// TIA Portal V17 export
// export: Created 2023-02-14T02:49:55.0959699Z, ExportSetting WithDefaults, DisplayName Totally Integrated Automation Portal, DisplayVersion V17, DisplayName TIA Portal Openness, DisplayVersion V17, DisplayName TIA Portal Teamcenter Gateway, DisplayVersion V17, DisplayName TIA Portal Version Control Interface, DisplayVersion V17, DisplayName SINAMICS Startdrive Advanced, DisplayVersion V17, DisplayName SINAMICS Startdrive G130, G150, S120, S150, SINAMICS MV, S210, DisplayVersion V17, DisplayName SINAMICS Startdrive G110M, G120, G120C, G120D, G120P, G115D, DisplayVersion V17, DisplayName STEP 7 Professional, DisplayVersion V17, DisplayName STEP 7 Safety, DisplayVersion V17, DisplayName WinCC Professional, DisplayVersion V17
VAR_GLOBAL   // PLC tag table "RIO Preparation"
   "FT-51.01" AT %IW83 : Int;
   "TT-51.01" AT %IW85 : Int;
   "LT-02.01" AT %IW87 : Int;
   "LT-03.01" AT %IW89 : Int;
   "LT-04.01" AT %IW91 : Int;
   "LT-05.01" AT %IW93 : Int;
   "LT-06.01" AT %IW95 : Int;
   "LT-07.01" AT %IW97 : Int;
   "LT-08.01" AT %IW99 : Int;
   "LT-09.01" AT %IW101 : Int;
   "LT-10.01" AT %IW103 : Int;
   "ZSC-51.04" AT %I75.0 : Bool;
   "ZSC-51.05" AT %I75.1 : Bool;
   "LL-51.01" AT %I75.2 : Bool;
   "ML-51.01" AT %I75.3 : Bool;
   "HL-51.01" AT %I75.4 : Bool;
   "ZSC-02.01" AT %I75.5 : Bool;
   "ZSC-02.02" AT %I75.6 : Bool;
   "ZSC-02.03" AT %I75.7 : Bool;
   "ZSC-02.04" AT %I76.0 : Bool;
   "ZSC-02.11" AT %I76.1 : Bool;
   "ZSC-02.12" AT %I76.2 : Bool;
   "ZSC-02.13" AT %I76.3 : Bool;
   "ZSC-03.01" AT %I76.4 : Bool;
   "ZSC-03.02" AT %I76.5 : Bool;
   "ZSC-03.03" AT %I76.6 : Bool;
   "ZSC-03.04" AT %I76.7 : Bool;
   "ZSC-03.06" AT %I77.0 : Bool;
   "ZSC-03.11" AT %I77.1 : Bool;
   "ZSC-03.12" AT %I77.2 : Bool;
   "ZSC-03.13" AT %I77.3 : Bool;
   "ZSC-04.01" AT %I77.4 : Bool;
   "ZSC-04.02" AT %I77.5 : Bool;
   "ZSC-04.03" AT %I77.6 : Bool;
   "ZSC-04.04" AT %I77.7 : Bool;
   "ZSC-04.06" AT %I78.0 : Bool;
   "ZSC-04.11" AT %I78.1 : Bool;
   "ZSC-04.12" AT %I78.2 : Bool;
   "ZSC-04.13" AT %I78.3 : Bool;
   "DRP-P02.01" AT %I78.4 : Bool;
   "DRP-P02.02" AT %I78.5 : Bool;
   "DRP-P03.01" AT %I78.6 : Bool;
   "DRP-P03.02" AT %I78.7 : Bool;
   "DRP-P04.01" AT %I79.0 : Bool;
   "ZSC-05.01" AT %I79.1 : Bool;
   "ZSC-05.02" AT %I79.2 : Bool;
   "ZSC-05.03" AT %I79.3 : Bool;
   "ZSC-05.04" AT %I79.4 : Bool;
   "ZSC-05.05" AT %I79.5 : Bool;
   "ZSC-05.06" AT %I79.6 : Bool;
   "ZSC-05.07" AT %I79.7 : Bool;
   "ZSC-05.09" AT %I80.0 : Bool;
   "ZSC-05.11" AT %I80.1 : Bool;
   "ZSC-05.12" AT %I80.2 : Bool;
   "ZSC-05.13" AT %I80.3 : Bool;
   "DRP-P05.01" AT %I80.4 : Bool;
   "DRP-P05.02" AT %I80.5 : Bool;
   "ZSC-06.01" AT %I80.6 : Bool;
   "ZSC-06.02" AT %I80.7 : Bool;
   "ZSC-06.03" AT %I81.0 : Bool;
   "ZSC-06.04" AT %I81.1 : Bool;
   "ZSC-06.11" AT %I81.2 : Bool;
   "ZSC-06.12" AT %I81.3 : Bool;
   "ZSC-06.13" AT %I81.4 : Bool;
   "ZSC-07.01" AT %I81.5 : Bool;
   "ZSC-07.02" AT %I81.6 : Bool;
   "ZSC-07.03" AT %I81.7 : Bool;
   "ZSC-07.04" AT %I82.0 : Bool;
   "ZSC-07.11" AT %I82.1 : Bool;
   "ZSC-07.12" AT %I82.2 : Bool;
   "ZSC-07.13" AT %I82.3 : Bool;
   "ZSC-08.01" AT %I82.4 : Bool;
   "ZSC-08.02" AT %I82.5 : Bool;
   "ZSC-08.03" AT %I82.6 : Bool;
   "ZSC-08.04" AT %I82.7 : Bool;
   "Spare Prep 2" AT %IW107 : Int;
   "Spare Prep 3" AT %IW109 : Int;
   "Spare Prep 4" AT %IW111 : Int;
   "Spare Prep 5" AT %IW113 : Int;
   "ZSC-08.11" AT %I671.0 : Bool;
   "ZSC-08.12" AT %I671.1 : Bool;
   "ZSC-08.13" AT %I671.2 : Bool;
   "ZSC-08.14" AT %I671.3 : Bool;
   "ZSC-08.15" AT %I671.4 : Bool;
   "DRP-P06.01" AT %I671.5 : Bool;
   "DRP-P07.01" AT %I671.6 : Bool;
   "DRP-P08.01" AT %I671.7 : Bool;
   "ZSC-09.01" AT %I672.0 : Bool;
   "ZSC-09.02" AT %I672.1 : Bool;
   "ZSC-09.03" AT %I672.2 : Bool;
   "ZSC-09.04" AT %I672.3 : Bool;
   "ZSC-09.05" AT %I672.4 : Bool;
   "ZSC-09.11" AT %I672.5 : Bool;
   "ZSC-09.12" AT %I672.6 : Bool;
   "ZSC-09.13" AT %I672.7 : Bool;
   "ZSC-10.02" AT %I673.0 : Bool;
   "DRP-P09.01" AT %I673.1 : Bool;
   "DRP-P09.02" AT %I673.2 : Bool;
   "EM STOP RIO PREPARATION" AT %I673.3 : Bool;
   "PS-01 Valve Terminal 1 Prep" AT %I673.4 : Bool;
   "ES1-P05.03" AT %I673.5 : Bool;
   "PB1-P05.03" AT %I673.6 : Bool;
   "PB2-P05.03" AT %I673.7 : Bool;
   "ES1-P09.03" AT %I674.0 : Bool;
   "PB1-P09.03" AT %I674.1 : Bool;
   "PB2-P09.03" AT %I674.2 : Bool;
   "ES1-P10.02" AT %I674.3 : Bool;
   "PB1-P10.02" AT %I674.4 : Bool;
   "PB2-P10.02" AT %I674.5 : Bool;
   "Pulse FT-51.01" AT %I675.0 : Bool;
   "Spare Prep 1" AT %IW105 : Int;
   "Spare Prep 15" AT %I674.6 : Bool;
   "Spare Prep 16" AT %I674.7 : Bool;
   "Spare Prep 17" AT %I675.1 : Bool;
   "Spare Prep 18" AT %I675.2 : Bool;
   "Spare Prep 19" AT %I675.3 : Bool;
   "Spare Prep 20" AT %I675.4 : Bool;
   "Spare Prep 21" AT %I675.5 : Bool;
   "Spare Prep 22" AT %I675.6 : Bool;
   "Spare Prep 23" AT %I675.7 : Bool;
   "SV-10.01 / P-10.02" AT %Q9.0 : Bool;
   "P-05.03 ON STATUS FEEDING PUMP" AT %Q9.1 : Bool;
   "CV-51.11" AT %QW12 : Int;
   "AV-51.01" AT %Q46.0 : Bool;
   "AV-51.02" AT %Q46.1 : Bool;
   "AV-51.03" AT %Q46.2 : Bool;
   "AV-51.04" AT %Q46.3 : Bool;
   "AV-51.05" AT %Q46.4 : Bool;
   "AV-02.01" AT %Q46.5 : Bool;
   "AV-02.02" AT %Q46.6 : Bool;
   "AV-02.03" AT %Q46.7 : Bool;
   "AV-02.04" AT %Q47.0 : Bool;
   "AV-02.05" AT %Q47.1 : Bool;
   "AV-02.06" AT %Q47.2 : Bool;
   "AV-02.10" AT %Q47.3 : Bool;
   "AV-02.11" AT %Q47.4 : Bool;
   "AV-02.12" AT %Q47.5 : Bool;
   "AV-02.13" AT %Q47.6 : Bool;
   "AV-02.20" AT %Q47.7 : Bool;
   "AV-03.01" AT %Q48.0 : Bool;
   "AV-03.02" AT %Q48.1 : Bool;
   "AV-03.03" AT %Q48.2 : Bool;
   "AV-03.04" AT %Q48.3 : Bool;
   "AV-03.05" AT %Q48.4 : Bool;
   "AV-03.06" AT %Q48.5 : Bool;
   "AV-03.10" AT %Q48.6 : Bool;
   "AV-03.11" AT %Q48.7 : Bool;
   "AV-03.12" AT %Q49.0 : Bool;
   "AV-03.13" AT %Q49.1 : Bool;
   "AV-04.01" AT %Q49.2 : Bool;
   "AV-04.02" AT %Q49.3 : Bool;
   "AV-04.03" AT %Q49.4 : Bool;
   "AV-04.04" AT %Q49.5 : Bool;
   "AV-04.05" AT %Q49.6 : Bool;
   "AV-04.06" AT %Q49.7 : Bool;
   "AV-04.10" AT %Q50.0 : Bool;
   "AV-04.11" AT %Q50.1 : Bool;
   "AV-04.12" AT %Q50.2 : Bool;
   "AV-04.13" AT %Q50.3 : Bool;
   "AV-05.01" AT %Q50.4 : Bool;
   "AV-05.02" AT %Q50.5 : Bool;
   "AV-05.03" AT %Q50.6 : Bool;
   "AV-05.04" AT %Q50.7 : Bool;
   "AV-05.05" AT %Q51.0 : Bool;
   "AV-05.06" AT %Q51.1 : Bool;
   "AV-05.07" AT %Q51.2 : Bool;
   "AV-05.08" AT %Q51.3 : Bool;
   "AV-05.09" AT %Q51.4 : Bool;
   "AV-05.10" AT %Q51.5 : Bool;
   "AV-05.11" AT %Q51.6 : Bool;
   "AV-05.12" AT %Q51.7 : Bool;
   "P-09.03 ON STATUS FEEDING PUMP" AT %Q9.2 : Bool;
   "P-10.02 ON STATUS FEEDING PUMP" AT %Q9.3 : Bool;
   "DRP-P02.01 Switching Input" AT %Q9.4 : Bool;
   "DRP-P02.02 Switching Input" AT %Q9.5 : Bool;
   "DRP-P03.01 Switching Input" AT %Q9.6 : Bool;
   "DRP-P03.02 Switching Input" AT %Q9.7 : Bool;
   "DRP-P04.01 Switching Input" AT %Q10.0 : Bool;
   "DRP-P05.01 Switching Input" AT %Q10.1 : Bool;
   "DRP-P05.02 Switching Input" AT %Q10.2 : Bool;
   "DRP-P06.01 Switching Input" AT %Q10.3 : Bool;
   "DRP-P07.01 Switching Input" AT %Q10.4 : Bool;
   "DRP-P08.01 Switching Input" AT %Q10.5 : Bool;
   "DRP-P09.01 Switching Input" AT %Q10.6 : Bool;
   "DRP-P09.02 Switching Input" AT %Q10.7 : Bool;
   "Spare Prep 7" AT %Q11.0 : Bool;
   "Spare Prep 8" AT %Q11.1 : Bool;
   "Spare Prep 9" AT %Q11.2 : Bool;
   "Spare Prep 10" AT %Q11.3 : Bool;
   "Spare Prep 11" AT %Q11.4 : Bool;
   "Spare Prep 12" AT %Q11.5 : Bool;
   "Spare Prep 13" AT %Q11.6 : Bool;
   "Spare Prep 14" AT %Q11.7 : Bool;
   "Spare Prep 6" AT %QW14 : Int;
   "AV-05.13" AT %Q52.0 : Bool;
   "AV-05.14" AT %Q52.1 : Bool;
   "AV-05.20" AT %Q52.2 : Bool;
   "AV-06.01" AT %Q52.3 : Bool;
   "AV-06.02" AT %Q52.4 : Bool;
   "AV-06.03" AT %Q52.5 : Bool;
   "AV-06.04" AT %Q52.6 : Bool;
   "AV-06.05" AT %Q52.7 : Bool;
   "AV-06.10" AT %Q53.0 : Bool;
   "AV-06.11" AT %Q53.1 : Bool;
   "AV-06.12" AT %Q53.2 : Bool;
   "AV-06.13" AT %Q53.3 : Bool;
   "AV-07.01" AT %Q53.4 : Bool;
   "AV-07.02" AT %Q53.5 : Bool;
   "AV-07.03" AT %Q53.6 : Bool;
   "AV-07.04" AT %Q53.7 : Bool;
   "AV-07.05" AT %Q68.0 : Bool;
   "AV-07.10" AT %Q68.1 : Bool;
   "AV-07.11" AT %Q68.2 : Bool;
   "AV-07.12" AT %Q68.3 : Bool;
   "AV-07.13" AT %Q68.4 : Bool;
   "AV-08.01" AT %Q68.5 : Bool;
   "AV-08.02" AT %Q68.6 : Bool;
   "AV-08.03" AT %Q68.7 : Bool;
   "AV-08.04" AT %Q69.0 : Bool;
   "AV-08.05" AT %Q69.1 : Bool;
   "AV-08.10" AT %Q69.2 : Bool;
   "AV-08.11" AT %Q69.3 : Bool;
   "AV-08.12" AT %Q69.4 : Bool;
   "AV-08.13" AT %Q69.5 : Bool;
   "AV-08.14" AT %Q69.6 : Bool;
   "AV-08.15" AT %Q69.7 : Bool;
   "AV-08.16" AT %Q70.0 : Bool;
   "AV-08.17" AT %Q70.1 : Bool;
   "AV-09.01" AT %Q70.2 : Bool;
   "AV-09.02" AT %Q70.3 : Bool;
   "AV-09.03" AT %Q70.4 : Bool;
   "AV-09.04" AT %Q70.5 : Bool;
   "AV-09.05" AT %Q70.6 : Bool;
   "AV-09.06" AT %Q70.7 : Bool;
   "AV-09.10" AT %Q71.0 : Bool;
   "AV-09.11" AT %Q71.1 : Bool;
   "AV-09.12" AT %Q71.2 : Bool;
   "AV-09.13" AT %Q71.3 : Bool;
   "AV-10.02" AT %Q71.4 : Bool;
   "AV-10.03" AT %Q71.5 : Bool;
END_VAR
